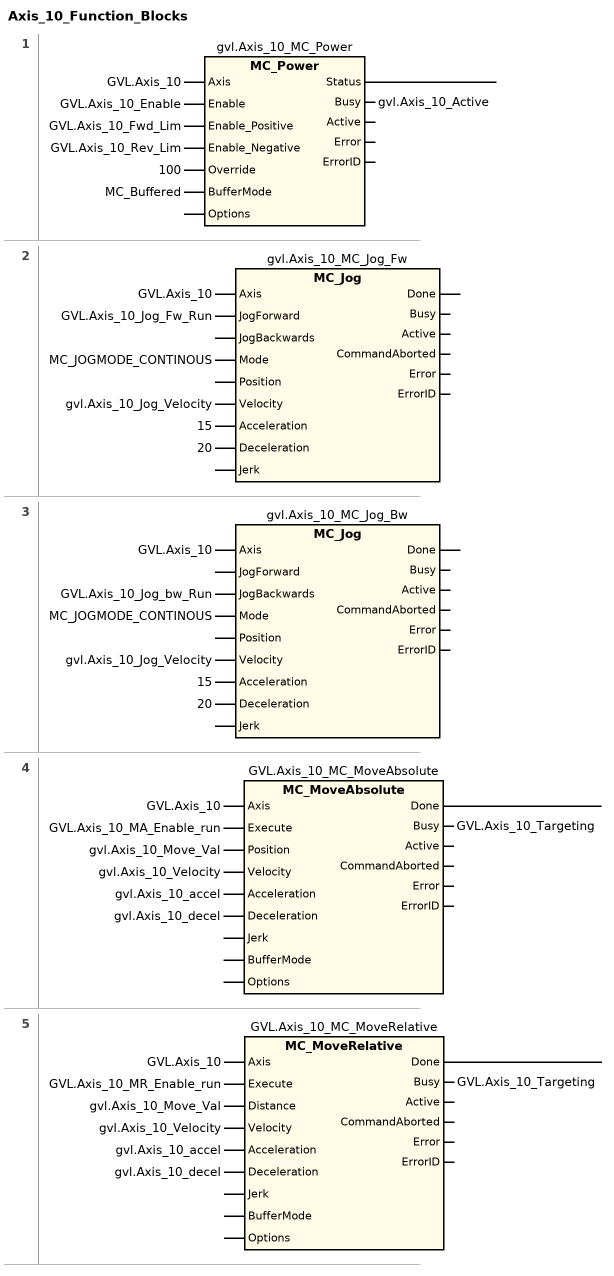
// NETWORK 1
gvl.Axis_10_MC_Power(
    Axis := GVL.Axis_10,
    Enable := GVL.Axis_10_Enable,
    Enable_Positive := GVL.Axis_10_Fwd_Lim,
    Enable_Negative := GVL.Axis_10_Rev_Lim,
    Override := 100,
    BufferMode := MC_Buffered,
    Busy => gvl.Axis_10_Active); // MC_Power

// NETWORK 2
gvl.Axis_10_MC_Jog_Fw(
    Axis := GVL.Axis_10,
    JogForward := GVL.Axis_10_Jog_Fw_Run,
    Mode := MC_JOGMODE_CONTINOUS,
    Velocity := gvl.Axis_10_Jog_Velocity,
    Acceleration := 15,
    Deceleration := 20); // MC_Jog

// NETWORK 3
gvl.Axis_10_MC_Jog_Bw(
    Axis := GVL.Axis_10,
    JogBackwards := GVL.Axis_10_Jog_bw_Run,
    Mode := MC_JOGMODE_CONTINOUS,
    Velocity := gvl.Axis_10_Jog_Velocity,
    Acceleration := 15,
    Deceleration := 20); // MC_Jog

// NETWORK 4
GVL.Axis_10_MC_MoveAbsolute(
    Axis := GVL.Axis_10,
    Execute := GVL.Axis_10_MA_Enable_run,
    Position := gvl.Axis_10_Move_Val,
    Velocity := gvl.Axis_10_Velocity,
    Acceleration := gvl.Axis_10_accel,
    Deceleration := gvl.Axis_10_decel,
    Busy => GVL.Axis_10_Targeting); // MC_MoveAbsolute

// NETWORK 5
GVL.Axis_10_MC_MoveRelative(
    Axis := GVL.Axis_10,
    Execute := GVL.Axis_10_MR_Enable_run,
    Distance := gvl.Axis_10_Move_Val,
    Velocity := gvl.Axis_10_Velocity,
    Acceleration := gvl.Axis_10_accel,
    Deceleration := gvl.Axis_10_decel,
    Busy => GVL.Axis_10_Targeting); // MC_MoveRelative

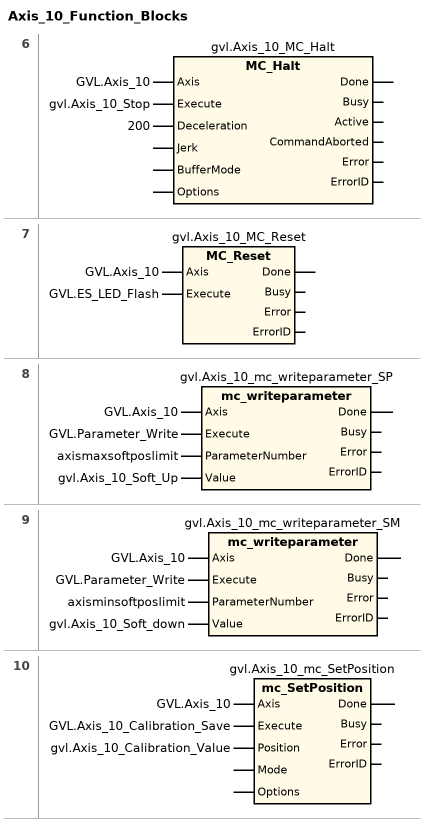
// NETWORK 6
gvl.Axis_10_MC_Halt(Axis := GVL.Axis_10, Execute := gvl.Axis_10_Stop, Deceleration := 200); // MC_Halt

// NETWORK 7
gvl.Axis_10_MC_Reset(Axis := GVL.Axis_10, Execute := GVL.ES_LED_Flash); // MC_Reset

// NETWORK 8
gvl.Axis_10_mc_writeparameter_SP(
    Axis := GVL.Axis_10,
    Execute := GVL.Parameter_Write,
    ParameterNumber := axismaxsoftposlimit,
    Value := gvl.Axis_10_Soft_Up); // mc_writeparameter

// NETWORK 9
gvl.Axis_10_mc_writeparameter_SM(
    Axis := GVL.Axis_10,
    Execute := GVL.Parameter_Write,
    ParameterNumber := axisminsoftposlimit,
    Value := gvl.Axis_10_Soft_down); // mc_writeparameter

// NETWORK 10
gvl.Axis_10_mc_SetPosition(
    Axis := GVL.Axis_10,
    Execute := GVL.Axis_10_Calibration_Save,
    Position := gvl.Axis_10_Calibration_Value); // mc_SetPosition

END_PROGRAM

// ---- POUs/Axis_10_Logic.TcPOU
PROGRAM Axis_10_Logic
VAR
	TON_0: TON;
	TON_1: TON;
	TON_2: TON;
	TON_3: TON;
	Axis_10_Velocity_Range: LREAL;
	Axis_10_Velocity_Scale: LREAL;
	Axis_10_Velocity_Raw: LREAL;
	Axis_10_Soft_Range: LREAL;
	Axis_10_Soft_Position: LREAL;
	Axis_10_Soft_Position_In_Range: LREAL;
END_VAR

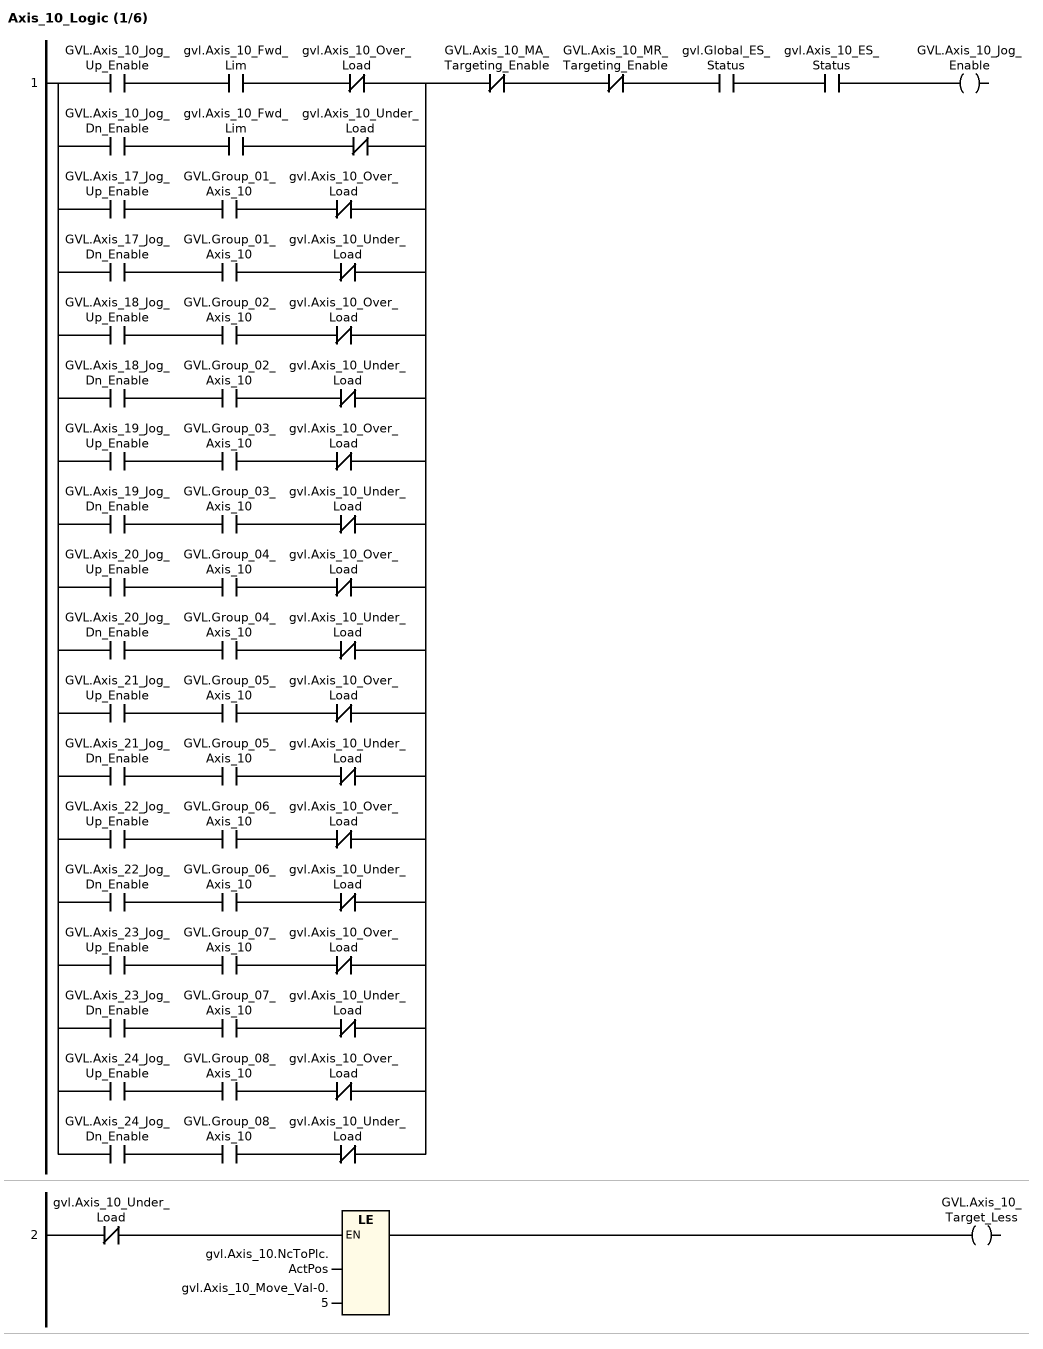
// NETWORK 1
GVL.Axis_10_Jog_Enable := (GVL.Axis_10_Jog_Up_Enable AND gvl.Axis_10_Fwd_Lim AND NOT gvl.Axis_10_Over_Load OR GVL.Axis_10_Jog_Dn_Enable AND gvl.Axis_10_Fwd_Lim AND NOT gvl.Axis_10_Under_Load OR GVL.Axis_17_Jog_Up_Enable AND GVL.Group_01_Axis_10 AND NOT gvl.Axis_10_Over_Load OR GVL.Axis_17_Jog_Dn_Enable AND GVL.Group_01_Axis_10 AND NOT gvl.Axis_10_Under_Load OR GVL.Axis_18_Jog_Up_Enable AND GVL.Group_02_Axis_10 AND NOT gvl.Axis_10_Over_Load OR GVL.Axis_18_Jog_Dn_Enable AND GVL.Group_02_Axis_10 AND NOT gvl.Axis_10_Under_Load OR GVL.Axis_19_Jog_Up_Enable AND GVL.Group_03_Axis_10 AND NOT gvl.Axis_10_Over_Load OR GVL.Axis_19_Jog_Dn_Enable AND GVL.Group_03_Axis_10 AND NOT gvl.Axis_10_Under_Load OR GVL.Axis_20_Jog_Up_Enable AND GVL.Group_04_Axis_10 AND NOT gvl.Axis_10_Over_Load OR GVL.Axis_20_Jog_Dn_Enable AND GVL.Group_04_Axis_10 AND NOT gvl.Axis_10_Under_Load OR GVL.Axis_21_Jog_Up_Enable AND GVL.Group_05_Axis_10 AND NOT gvl.Axis_10_Over_Load OR GVL.Axis_21_Jog_Dn_Enable AND GVL.Group_05_Axis_10 AND NOT gvl.Axis_10_Under_Load OR GVL.Axis_22_Jog_Up_Enable AND GVL.Group_06_Axis_10 AND NOT gvl.Axis_10_Over_Load OR GVL.Axis_22_Jog_Dn_Enable AND GVL.Group_06_Axis_10 AND NOT gvl.Axis_10_Under_Load OR GVL.Axis_23_Jog_Up_Enable AND GVL.Group_07_Axis_10 AND NOT gvl.Axis_10_Over_Load OR GVL.Axis_23_Jog_Dn_Enable AND GVL.Group_07_Axis_10 AND NOT gvl.Axis_10_Under_Load OR GVL.Axis_24_Jog_Up_Enable AND GVL.Group_08_Axis_10 AND NOT gvl.Axis_10_Over_Load OR GVL.Axis_24_Jog_Dn_Enable AND GVL.Group_08_Axis_10 AND NOT gvl.Axis_10_Under_Load) AND NOT GVL.Axis_10_MA_Targeting_Enable AND NOT GVL.Axis_10_MR_Targeting_Enable AND gvl.Global_ES_Status AND gvl.Axis_10_ES_Status;

// NETWORK 2
GVL.Axis_10_Target_Less := NOT gvl.Axis_10_Under_Load AND gvl.Axis_10.NcToPlc.ActPos <= (gvl.Axis_10_Move_Val-0.5);

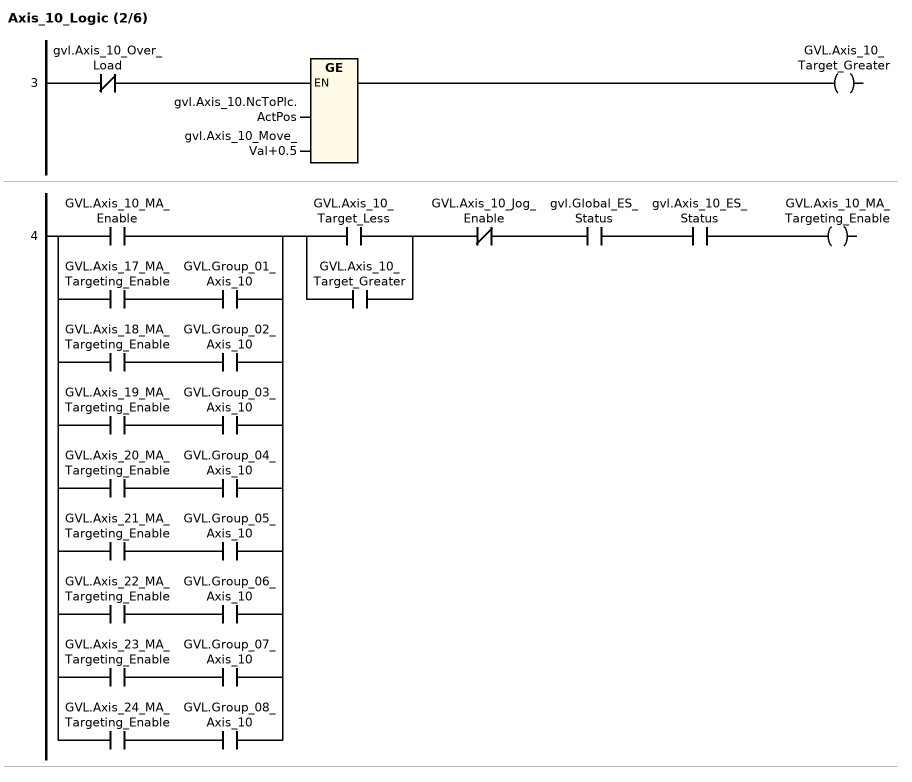
// NETWORK 3
GVL.Axis_10_Target_Greater := NOT gvl.Axis_10_Over_Load AND gvl.Axis_10.NcToPlc.ActPos >= (gvl.Axis_10_Move_Val+0.5);

// NETWORK 4
GVL.Axis_10_MA_Targeting_Enable := (GVL.Axis_10_MA_Enable OR GVL.Axis_17_MA_Targeting_Enable AND GVL.Group_01_Axis_10 OR GVL.Axis_18_MA_Targeting_Enable AND GVL.Group_02_Axis_10 OR GVL.Axis_19_MA_Targeting_Enable AND GVL.Group_03_Axis_10 OR GVL.Axis_20_MA_Targeting_Enable AND GVL.Group_04_Axis_10 OR GVL.Axis_21_MA_Targeting_Enable AND GVL.Group_05_Axis_10 OR GVL.Axis_22_MA_Targeting_Enable AND GVL.Group_06_Axis_10 OR GVL.Axis_23_MA_Targeting_Enable AND GVL.Group_07_Axis_10 OR GVL.Axis_24_MA_Targeting_Enable AND GVL.Group_08_Axis_10) AND (GVL.Axis_10_Target_Less OR GVL.Axis_10_Target_Greater) AND NOT GVL.Axis_10_Jog_Enable AND gvl.Global_ES_Status AND gvl.Axis_10_ES_Status;

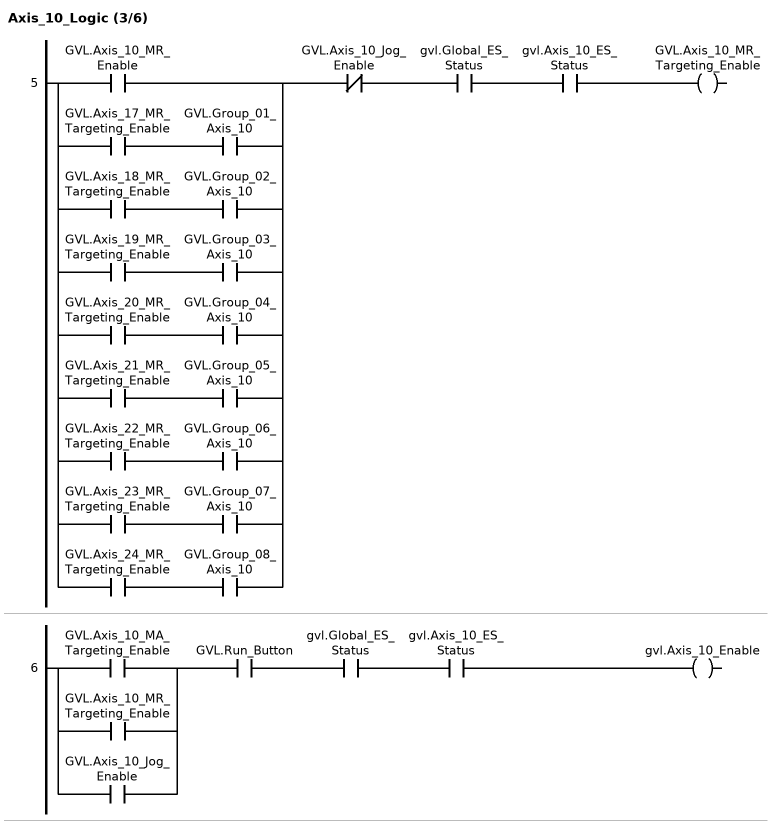
// NETWORK 5
GVL.Axis_10_MR_Targeting_Enable := (GVL.Axis_10_MR_Enable OR GVL.Axis_17_MR_Targeting_Enable AND GVL.Group_01_Axis_10 OR GVL.Axis_18_MR_Targeting_Enable AND GVL.Group_02_Axis_10 OR GVL.Axis_19_MR_Targeting_Enable AND GVL.Group_03_Axis_10 OR GVL.Axis_20_MR_Targeting_Enable AND GVL.Group_04_Axis_10 OR GVL.Axis_21_MR_Targeting_Enable AND GVL.Group_05_Axis_10 OR GVL.Axis_22_MR_Targeting_Enable AND GVL.Group_06_Axis_10 OR GVL.Axis_23_MR_Targeting_Enable AND GVL.Group_07_Axis_10 OR GVL.Axis_24_MR_Targeting_Enable AND GVL.Group_08_Axis_10) AND NOT GVL.Axis_10_Jog_Enable AND gvl.Global_ES_Status AND gvl.Axis_10_ES_Status;

// NETWORK 6
gvl.Axis_10_Enable := (GVL.Axis_10_MA_Targeting_Enable OR GVL.Axis_10_MR_Targeting_Enable OR GVL.Axis_10_Jog_Enable) AND GVL.Run_Button AND gvl.Global_ES_Status AND gvl.Axis_10_ES_Status;

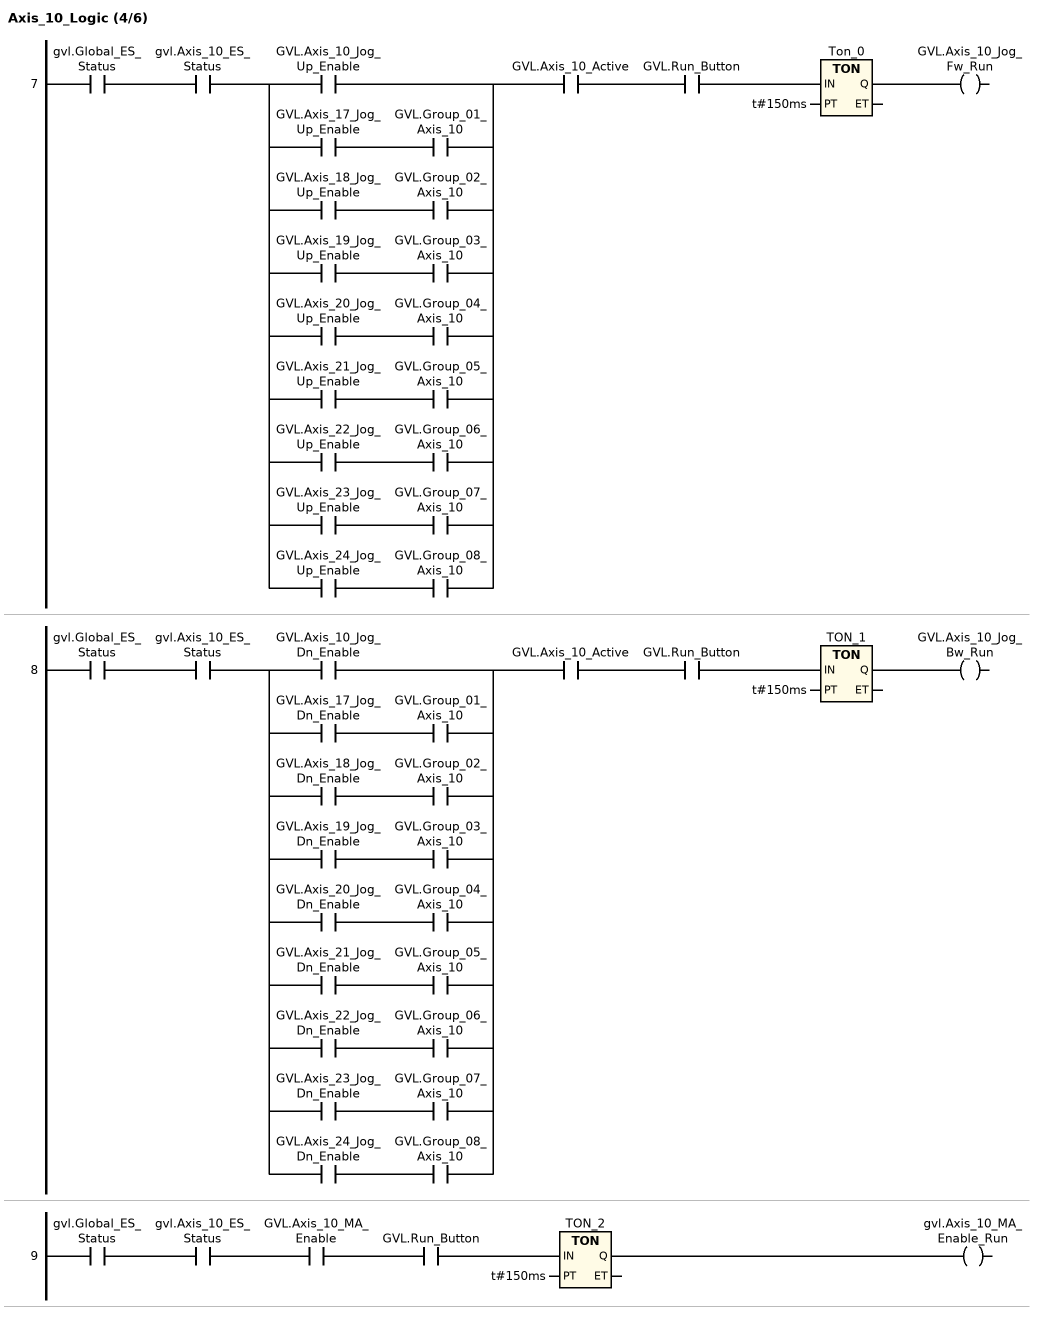
// NETWORK 7
Ton_0(IN := gvl.Global_ES_Status AND gvl.Axis_10_ES_Status AND (GVL.Axis_10_Jog_Up_Enable OR GVL.Axis_17_Jog_Up_Enable AND GVL.Group_01_Axis_10 OR GVL.Axis_18_Jog_Up_Enable AND GVL.Group_02_Axis_10 OR GVL.Axis_19_Jog_Up_Enable AND GVL.Group_03_Axis_10 OR GVL.Axis_20_Jog_Up_Enable AND GVL.Group_04_Axis_10 OR GVL.Axis_21_Jog_Up_Enable AND GVL.Group_05_Axis_10 OR GVL.Axis_22_Jog_Up_Enable AND GVL.Group_06_Axis_10 OR GVL.Axis_23_Jog_Up_Enable AND GVL.Group_07_Axis_10 OR GVL.Axis_24_Jog_Up_Enable AND GVL.Group_08_Axis_10) AND GVL.Axis_10_Active AND GVL.Run_Button, PT := t#150ms); // TON
GVL.Axis_10_Jog_Fw_Run := Ton_0.Q;

// NETWORK 8
TON_1(IN := gvl.Global_ES_Status AND gvl.Axis_10_ES_Status AND (GVL.Axis_10_Jog_Dn_Enable OR GVL.Axis_17_Jog_Dn_Enable AND GVL.Group_01_Axis_10 OR GVL.Axis_18_Jog_Dn_Enable AND GVL.Group_02_Axis_10 OR GVL.Axis_19_Jog_Dn_Enable AND GVL.Group_03_Axis_10 OR GVL.Axis_20_Jog_Dn_Enable AND GVL.Group_04_Axis_10 OR GVL.Axis_21_Jog_Dn_Enable AND GVL.Group_05_Axis_10 OR GVL.Axis_22_Jog_Dn_Enable AND GVL.Group_06_Axis_10 OR GVL.Axis_23_Jog_Dn_Enable AND GVL.Group_07_Axis_10 OR GVL.Axis_24_Jog_Dn_Enable AND GVL.Group_08_Axis_10) AND GVL.Axis_10_Active AND GVL.Run_Button, PT := t#150ms); // TON
GVL.Axis_10_Jog_Bw_Run := TON_1.Q;

// NETWORK 9
TON_2(IN := gvl.Global_ES_Status AND gvl.Axis_10_ES_Status AND GVL.Axis_10_MA_Enable AND GVL.Run_Button, PT := t#150ms); // TON
gvl.Axis_10_MA_Enable_Run := TON_2.Q;

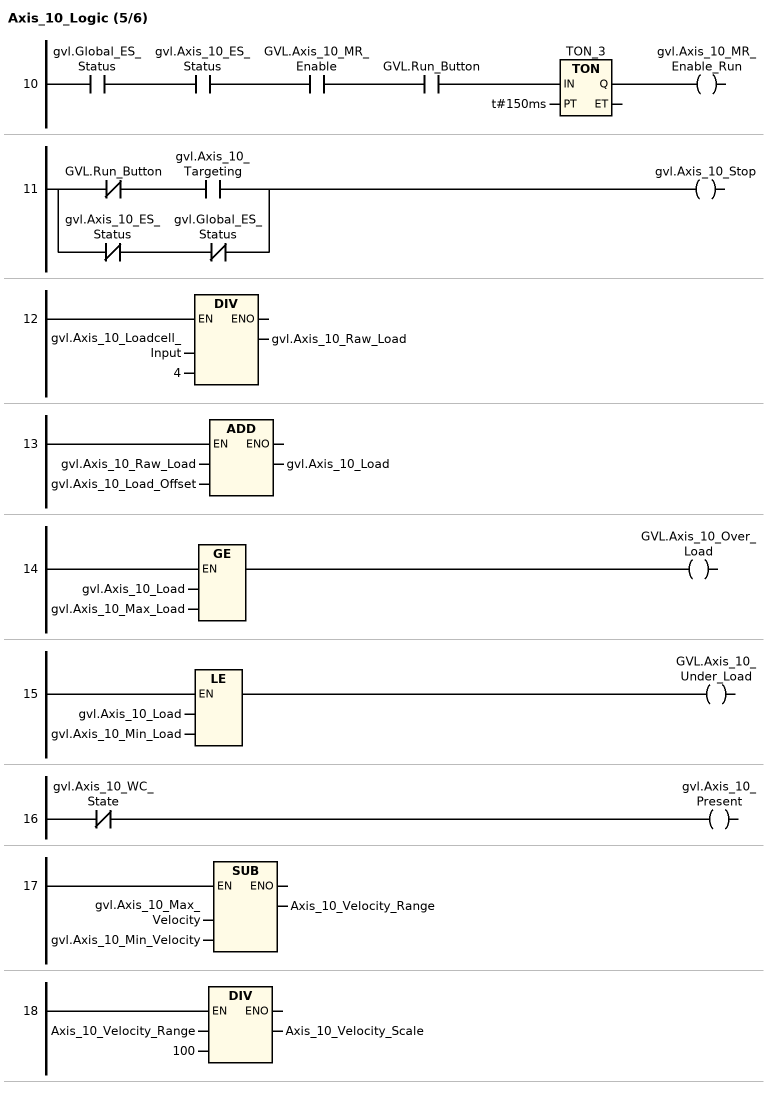
// NETWORK 10
TON_3(IN := gvl.Global_ES_Status AND gvl.Axis_10_ES_Status AND GVL.Axis_10_MR_Enable AND GVL.Run_Button, PT := t#150ms); // TON
gvl.Axis_10_MR_Enable_Run := TON_3.Q;

// NETWORK 11
gvl.Axis_10_Stop := NOT GVL.Run_Button AND gvl.Axis_10_Targeting OR NOT gvl.Axis_10_ES_Status AND NOT gvl.Global_ES_Status;

// NETWORK 12
gvl.Axis_10_Raw_Load := gvl.Axis_10_Loadcell_Input / 4;

// NETWORK 13
gvl.Axis_10_Load := gvl.Axis_10_Raw_Load + gvl.Axis_10_Load_Offset;

// NETWORK 14
GVL.Axis_10_Over_Load := gvl.Axis_10_Load >= gvl.Axis_10_Max_Load;

// NETWORK 15
GVL.Axis_10_Under_Load := gvl.Axis_10_Load <= gvl.Axis_10_Min_Load;

// NETWORK 16
gvl.Axis_10_Present := NOT gvl.Axis_10_WC_State;

// NETWORK 17
Axis_10_Velocity_Range := gvl.Axis_10_Max_Velocity - gvl.Axis_10_Min_Velocity;

// NETWORK 18
Axis_10_Velocity_Scale := Axis_10_Velocity_Range / 100;

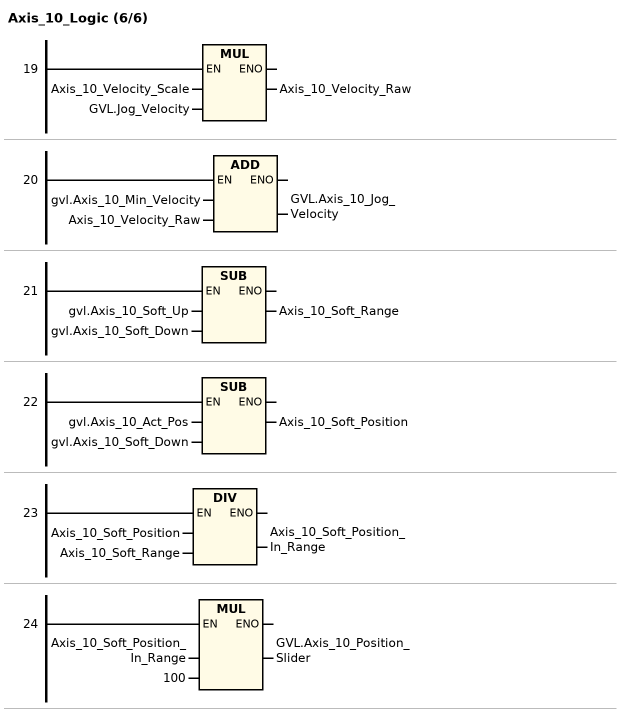
// NETWORK 19
Axis_10_Velocity_Raw := Axis_10_Velocity_Scale * GVL.Jog_Velocity;

// NETWORK 20
GVL.Axis_10_Jog_Velocity := gvl.Axis_10_Min_Velocity + Axis_10_Velocity_Raw;

// NETWORK 21
Axis_10_Soft_Range := gvl.Axis_10_Soft_Up - gvl.Axis_10_Soft_Down;

// NETWORK 22
Axis_10_Soft_Position := gvl.Axis_10_Act_Pos - gvl.Axis_10_Soft_Down;

// NETWORK 23
Axis_10_Soft_Position_In_Range := Axis_10_Soft_Position / Axis_10_Soft_Range;

// NETWORK 24
GVL.Axis_10_Position_Slider := Axis_10_Soft_Position_In_Range * 100;

END_PROGRAM

// ---- POUs/Axis_11_Function_Blocks.TcPOU
PROGRAM Axis_11_Function_Blocks
VAR
END_VAR

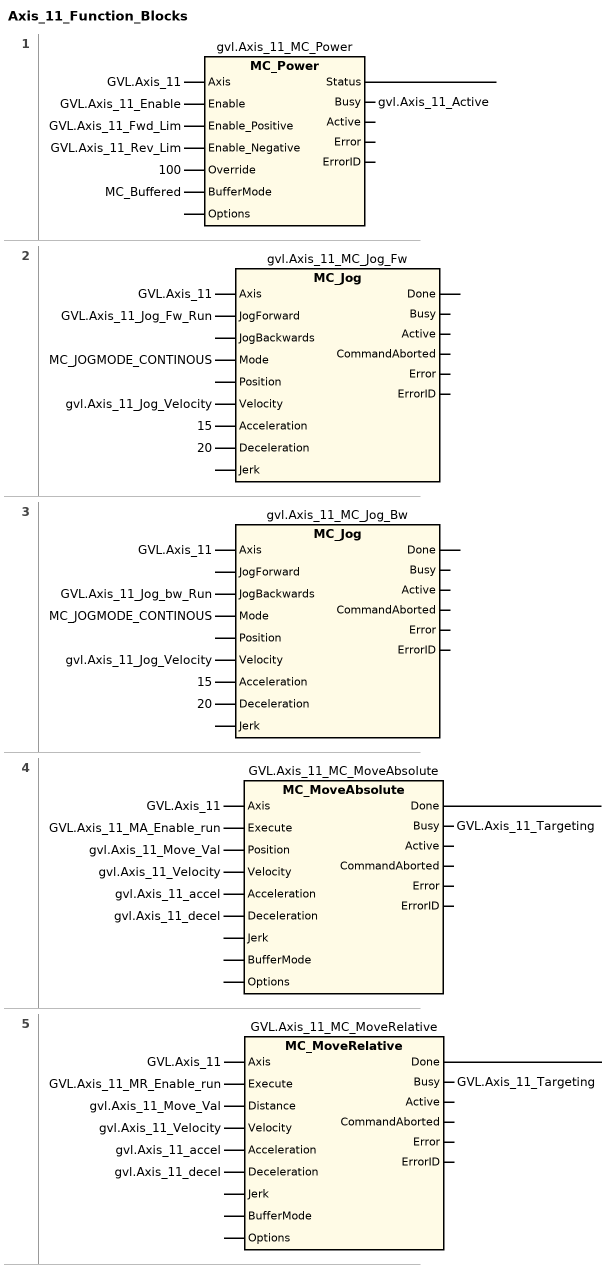
// NETWORK 1
gvl.Axis_11_MC_Power(
    Axis := GVL.Axis_11,
    Enable := GVL.Axis_11_Enable,
    Enable_Positive := GVL.Axis_11_Fwd_Lim,
    Enable_Negative := GVL.Axis_11_Rev_Lim,
    Override := 100,
    BufferMode := MC_Buffered,
    Busy => gvl.Axis_11_Active); // MC_Power

// NETWORK 2
gvl.Axis_11_MC_Jog_Fw(
    Axis := GVL.Axis_11,
    JogForward := GVL.Axis_11_Jog_Fw_Run,
    Mode := MC_JOGMODE_CONTINOUS,
    Velocity := gvl.Axis_11_Jog_Velocity,
    Acceleration := 15,
    Deceleration := 20); // MC_Jog

// NETWORK 3
gvl.Axis_11_MC_Jog_Bw(
    Axis := GVL.Axis_11,
    JogBackwards := GVL.Axis_11_Jog_bw_Run,
    Mode := MC_JOGMODE_CONTINOUS,
    Velocity := gvl.Axis_11_Jog_Velocity,
    Acceleration := 15,
    Deceleration := 20); // MC_Jog

// NETWORK 4
GVL.Axis_11_MC_MoveAbsolute(
    Axis := GVL.Axis_11,
    Execute := GVL.Axis_11_MA_Enable_run,
    Position := gvl.Axis_11_Move_Val,
    Velocity := gvl.Axis_11_Velocity,
    Acceleration := gvl.Axis_11_accel,
    Deceleration := gvl.Axis_11_decel,
    Busy => GVL.Axis_11_Targeting); // MC_MoveAbsolute

// NETWORK 5
GVL.Axis_11_MC_MoveRelative(
    Axis := GVL.Axis_11,
    Execute := GVL.Axis_11_MR_Enable_run,
    Distance := gvl.Axis_11_Move_Val,
    Velocity := gvl.Axis_11_Velocity,
    Acceleration := gvl.Axis_11_accel,
    Deceleration := gvl.Axis_11_decel,
    Busy => GVL.Axis_11_Targeting); // MC_MoveRelative

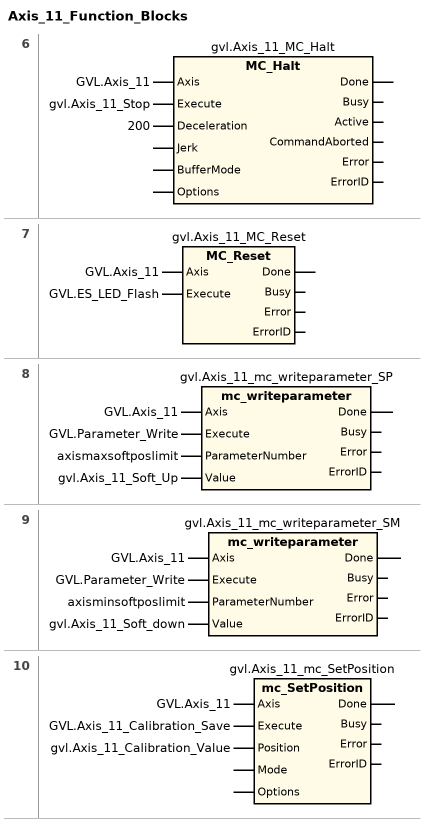
// NETWORK 6
gvl.Axis_11_MC_Halt(Axis := GVL.Axis_11, Execute := gvl.Axis_11_Stop, Deceleration := 200); // MC_Halt

// NETWORK 7
gvl.Axis_11_MC_Reset(Axis := GVL.Axis_11, Execute := GVL.ES_LED_Flash); // MC_Reset

// NETWORK 8
gvl.Axis_11_mc_writeparameter_SP(
    Axis := GVL.Axis_11,
    Execute := GVL.Parameter_Write,
    ParameterNumber := axismaxsoftposlimit,
    Value := gvl.Axis_11_Soft_Up); // mc_writeparameter

// NETWORK 9
gvl.Axis_11_mc_writeparameter_SM(
    Axis := GVL.Axis_11,
    Execute := GVL.Parameter_Write,
    ParameterNumber := axisminsoftposlimit,
    Value := gvl.Axis_11_Soft_down); // mc_writeparameter

// NETWORK 10
gvl.Axis_11_mc_SetPosition(
    Axis := GVL.Axis_11,
    Execute := GVL.Axis_11_Calibration_Save,
    Position := gvl.Axis_11_Calibration_Value); // mc_SetPosition

END_PROGRAM

// ---- POUs/Axis_11_Logic.TcPOU
PROGRAM Axis_11_Logic
VAR
	TON_0: TON;
	TON_1: TON;
	TON_2: TON;
	TON_3: TON;
	Axis_11_Velocity_Range: LREAL;
	Axis_11_Velocity_Scale: LREAL;
	Axis_11_Velocity_Raw: LREAL;
	Axis_11_Soft_Range: LREAL;
	Axis_11_Soft_Position: LREAL;
	Axis_11_Soft_Position_In_Range: LREAL;
END_VAR

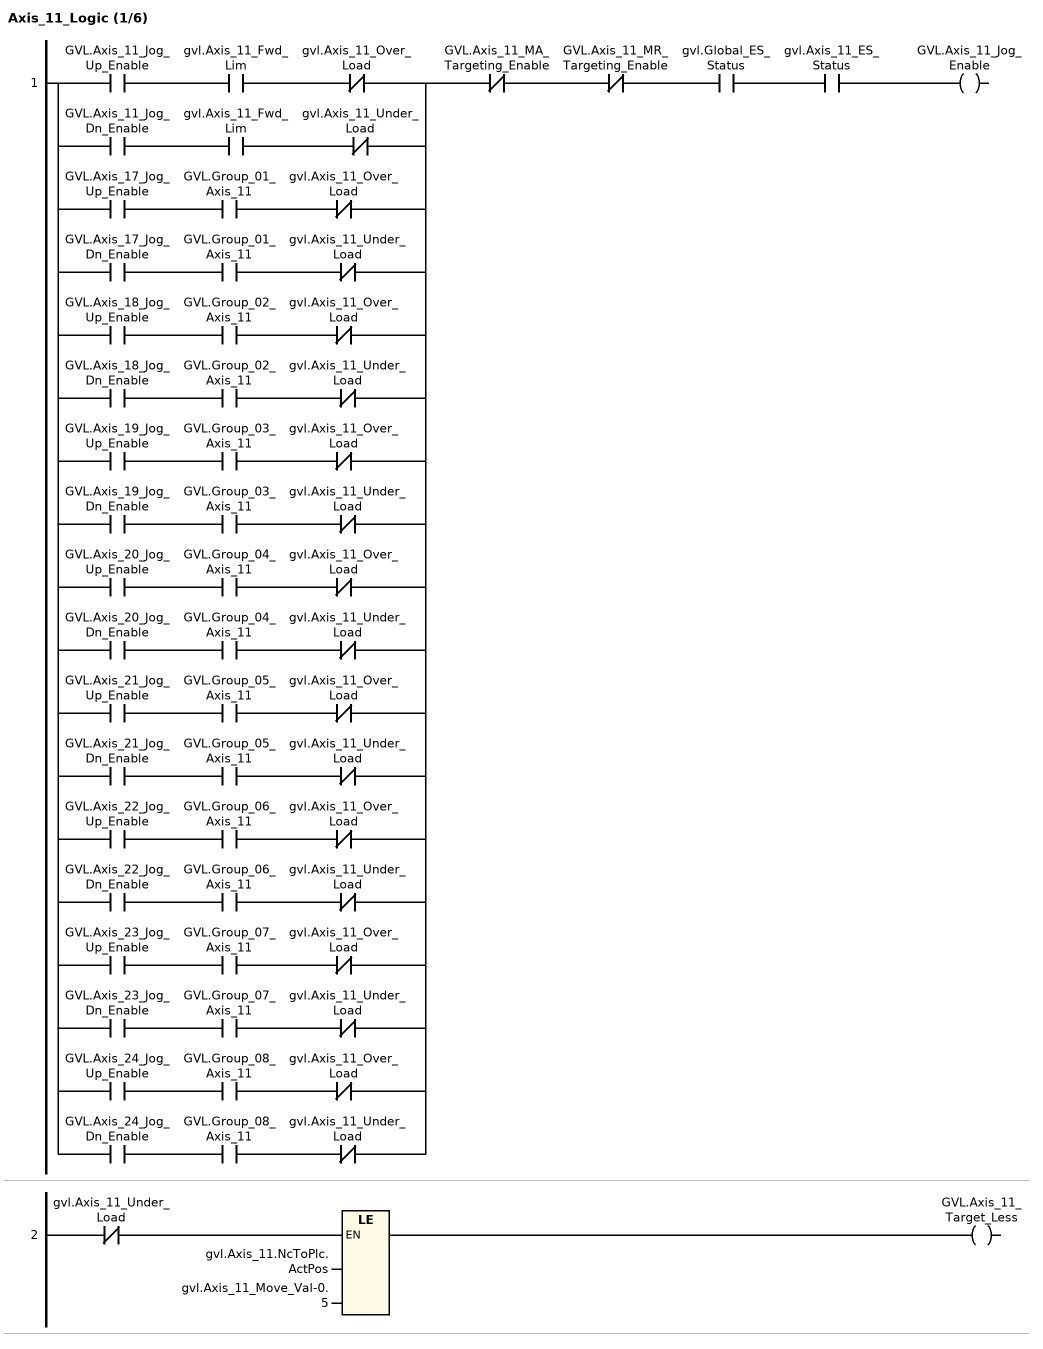
// NETWORK 1
GVL.Axis_11_Jog_Enable := (GVL.Axis_11_Jog_Up_Enable AND gvl.Axis_11_Fwd_Lim AND NOT gvl.Axis_11_Over_Load OR GVL.Axis_11_Jog_Dn_Enable AND gvl.Axis_11_Fwd_Lim AND NOT gvl.Axis_11_Under_Load OR GVL.Axis_17_Jog_Up_Enable AND GVL.Group_01_Axis_11 AND NOT gvl.Axis_11_Over_Load OR GVL.Axis_17_Jog_Dn_Enable AND GVL.Group_01_Axis_11 AND NOT gvl.Axis_11_Under_Load OR GVL.Axis_18_Jog_Up_Enable AND GVL.Group_02_Axis_11 AND NOT gvl.Axis_11_Over_Load OR GVL.Axis_18_Jog_Dn_Enable AND GVL.Group_02_Axis_11 AND NOT gvl.Axis_11_Under_Load OR GVL.Axis_19_Jog_Up_Enable AND GVL.Group_03_Axis_11 AND NOT gvl.Axis_11_Over_Load OR GVL.Axis_19_Jog_Dn_Enable AND GVL.Group_03_Axis_11 AND NOT gvl.Axis_11_Under_Load OR GVL.Axis_20_Jog_Up_Enable AND GVL.Group_04_Axis_11 AND NOT gvl.Axis_11_Over_Load OR GVL.Axis_20_Jog_Dn_Enable AND GVL.Group_04_Axis_11 AND NOT gvl.Axis_11_Under_Load OR GVL.Axis_21_Jog_Up_Enable AND GVL.Group_05_Axis_11 AND NOT gvl.Axis_11_Over_Load OR GVL.Axis_21_Jog_Dn_Enable AND GVL.Group_05_Axis_11 AND NOT gvl.Axis_11_Under_Load OR GVL.Axis_22_Jog_Up_Enable AND GVL.Group_06_Axis_11 AND NOT gvl.Axis_11_Over_Load OR GVL.Axis_22_Jog_Dn_Enable AND GVL.Group_06_Axis_11 AND NOT gvl.Axis_11_Under_Load OR GVL.Axis_23_Jog_Up_Enable AND GVL.Group_07_Axis_11 AND NOT gvl.Axis_11_Over_Load OR GVL.Axis_23_Jog_Dn_Enable AND GVL.Group_07_Axis_11 AND NOT gvl.Axis_11_Under_Load OR GVL.Axis_24_Jog_Up_Enable AND GVL.Group_08_Axis_11 AND NOT gvl.Axis_11_Over_Load OR GVL.Axis_24_Jog_Dn_Enable AND GVL.Group_08_Axis_11 AND NOT gvl.Axis_11_Under_Load) AND NOT GVL.Axis_11_MA_Targeting_Enable AND NOT GVL.Axis_11_MR_Targeting_Enable AND gvl.Global_ES_Status AND gvl.Axis_11_ES_Status;

// NETWORK 2
GVL.Axis_11_Target_Less := NOT gvl.Axis_11_Under_Load AND gvl.Axis_11.NcToPlc.ActPos <= (gvl.Axis_11_Move_Val-0.5);

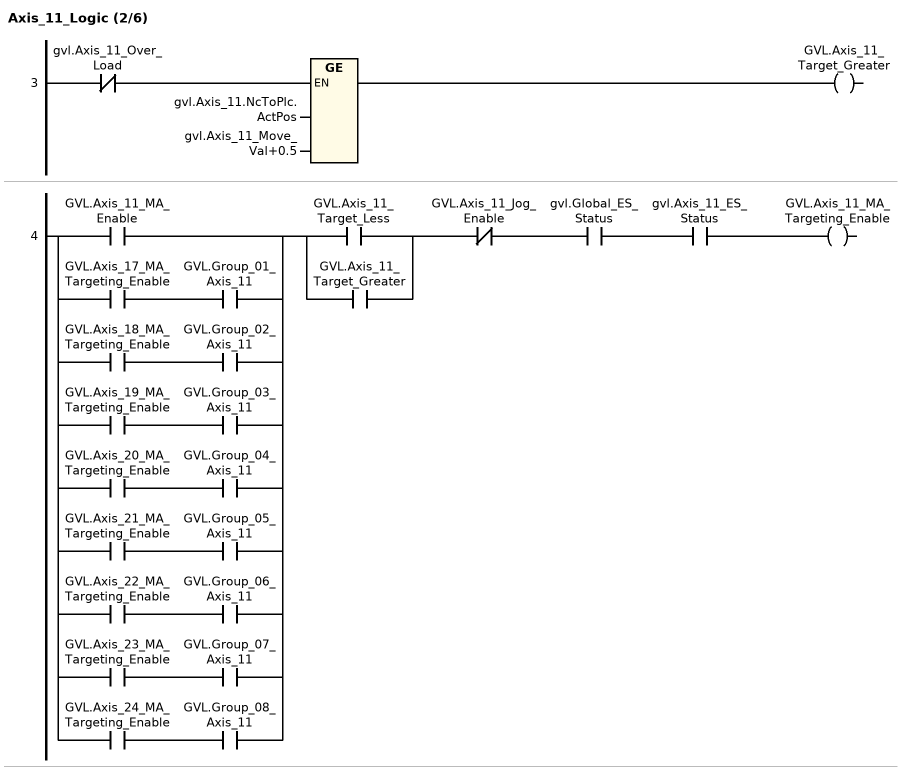
// NETWORK 3
GVL.Axis_11_Target_Greater := NOT gvl.Axis_11_Over_Load AND gvl.Axis_11.NcToPlc.ActPos >= (gvl.Axis_11_Move_Val+0.5);

// NETWORK 4
GVL.Axis_11_MA_Targeting_Enable := (GVL.Axis_11_MA_Enable OR GVL.Axis_17_MA_Targeting_Enable AND GVL.Group_01_Axis_11 OR GVL.Axis_18_MA_Targeting_Enable AND GVL.Group_02_Axis_11 OR GVL.Axis_19_MA_Targeting_Enable AND GVL.Group_03_Axis_11 OR GVL.Axis_20_MA_Targeting_Enable AND GVL.Group_04_Axis_11 OR GVL.Axis_21_MA_Targeting_Enable AND GVL.Group_05_Axis_11 OR GVL.Axis_22_MA_Targeting_Enable AND GVL.Group_06_Axis_11 OR GVL.Axis_23_MA_Targeting_Enable AND GVL.Group_07_Axis_11 OR GVL.Axis_24_MA_Targeting_Enable AND GVL.Group_08_Axis_11) AND (GVL.Axis_11_Target_Less OR GVL.Axis_11_Target_Greater) AND NOT GVL.Axis_11_Jog_Enable AND gvl.Global_ES_Status AND gvl.Axis_11_ES_Status;

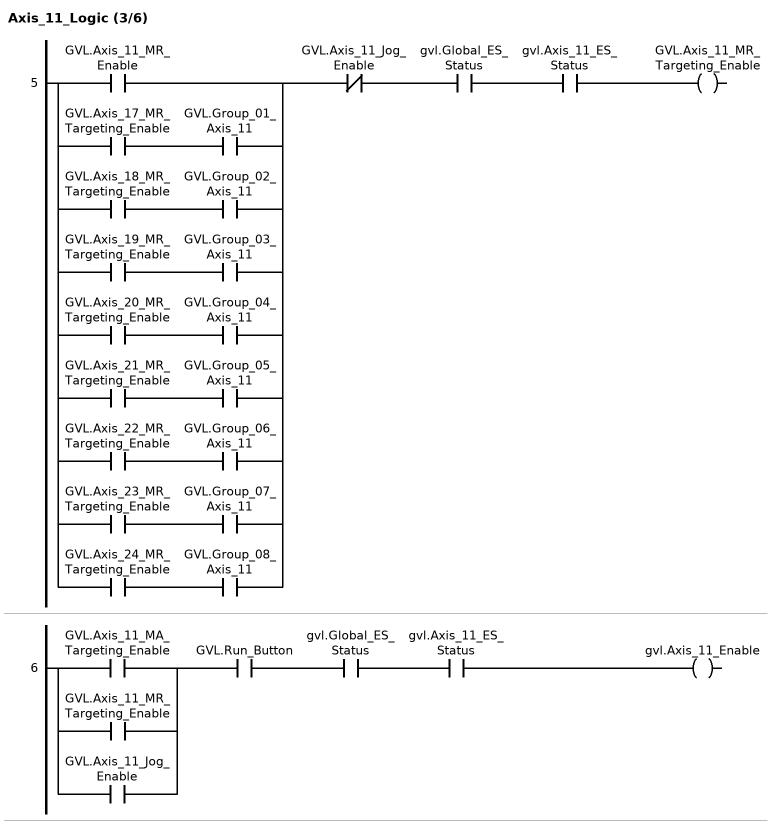
// NETWORK 5
GVL.Axis_11_MR_Targeting_Enable := (GVL.Axis_11_MR_Enable OR GVL.Axis_17_MR_Targeting_Enable AND GVL.Group_01_Axis_11 OR GVL.Axis_18_MR_Targeting_Enable AND GVL.Group_02_Axis_11 OR GVL.Axis_19_MR_Targeting_Enable AND GVL.Group_03_Axis_11 OR GVL.Axis_20_MR_Targeting_Enable AND GVL.Group_04_Axis_11 OR GVL.Axis_21_MR_Targeting_Enable AND GVL.Group_05_Axis_11 OR GVL.Axis_22_MR_Targeting_Enable AND GVL.Group_06_Axis_11 OR GVL.Axis_23_MR_Targeting_Enable AND GVL.Group_07_Axis_11 OR GVL.Axis_24_MR_Targeting_Enable AND GVL.Group_08_Axis_11) AND NOT GVL.Axis_11_Jog_Enable AND gvl.Global_ES_Status AND gvl.Axis_11_ES_Status;

// NETWORK 6
gvl.Axis_11_Enable := (GVL.Axis_11_MA_Targeting_Enable OR GVL.Axis_11_MR_Targeting_Enable OR GVL.Axis_11_Jog_Enable) AND GVL.Run_Button AND gvl.Global_ES_Status AND gvl.Axis_11_ES_Status;

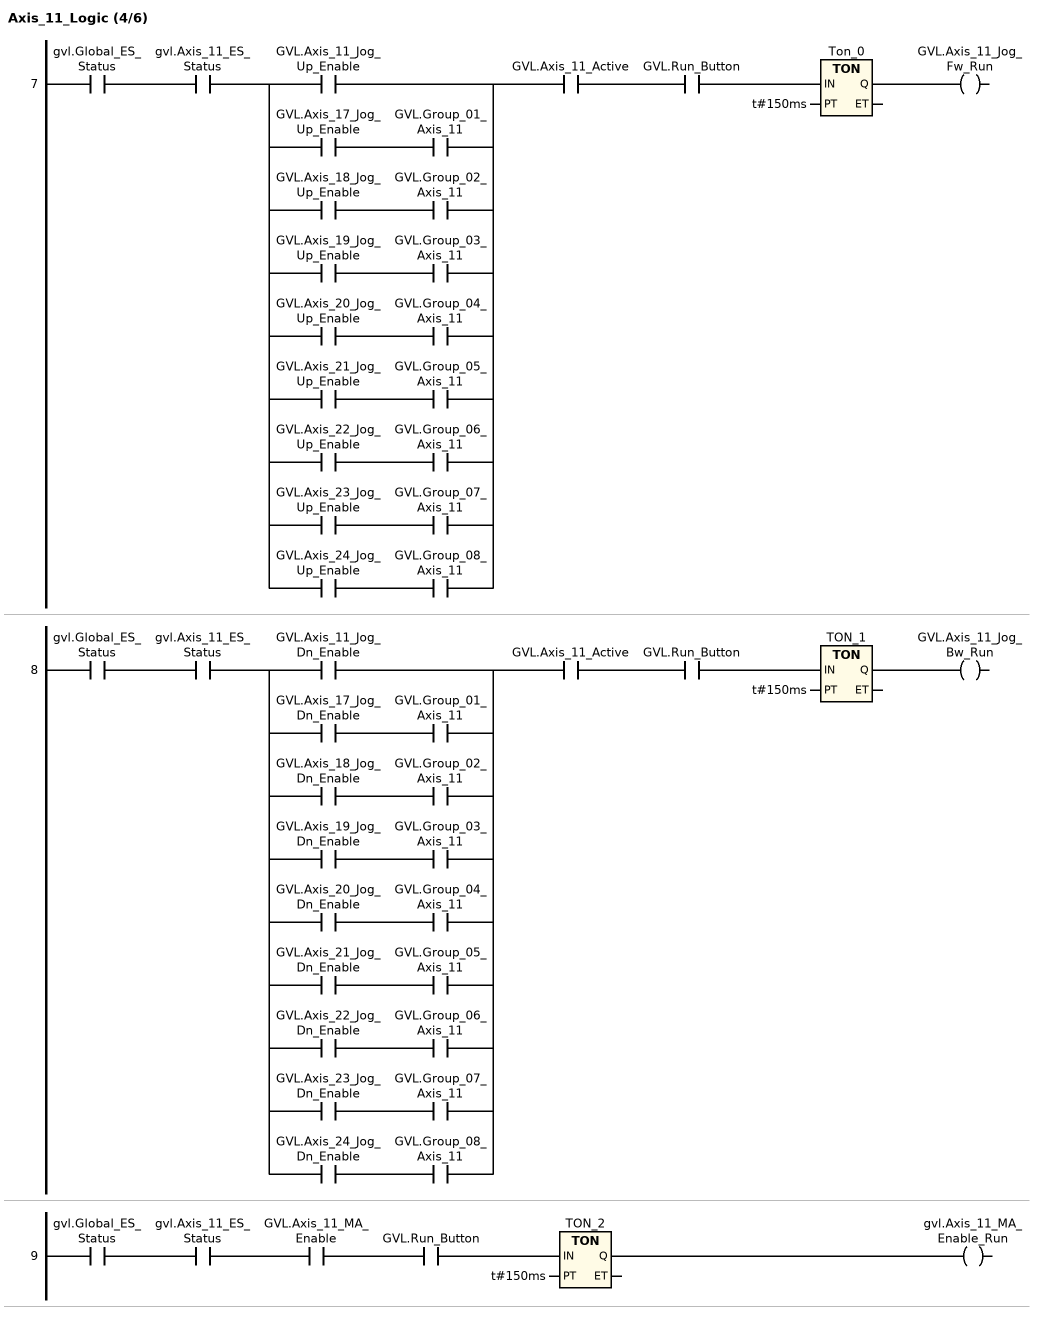
// NETWORK 7
Ton_0(IN := gvl.Global_ES_Status AND gvl.Axis_11_ES_Status AND (GVL.Axis_11_Jog_Up_Enable OR GVL.Axis_17_Jog_Up_Enable AND GVL.Group_01_Axis_11 OR GVL.Axis_18_Jog_Up_Enable AND GVL.Group_02_Axis_11 OR GVL.Axis_19_Jog_Up_Enable AND GVL.Group_03_Axis_11 OR GVL.Axis_20_Jog_Up_Enable AND GVL.Group_04_Axis_11 OR GVL.Axis_21_Jog_Up_Enable AND GVL.Group_05_Axis_11 OR GVL.Axis_22_Jog_Up_Enable AND GVL.Group_06_Axis_11 OR GVL.Axis_23_Jog_Up_Enable AND GVL.Group_07_Axis_11 OR GVL.Axis_24_Jog_Up_Enable AND GVL.Group_08_Axis_11) AND GVL.Axis_11_Active AND GVL.Run_Button, PT := t#150ms); // TON
GVL.Axis_11_Jog_Fw_Run := Ton_0.Q;

// NETWORK 8
TON_1(IN := gvl.Global_ES_Status AND gvl.Axis_11_ES_Status AND (GVL.Axis_11_Jog_Dn_Enable OR GVL.Axis_17_Jog_Dn_Enable AND GVL.Group_01_Axis_11 OR GVL.Axis_18_Jog_Dn_Enable AND GVL.Group_02_Axis_11 OR GVL.Axis_19_Jog_Dn_Enable AND GVL.Group_03_Axis_11 OR GVL.Axis_20_Jog_Dn_Enable AND GVL.Group_04_Axis_11 OR GVL.Axis_21_Jog_Dn_Enable AND GVL.Group_05_Axis_11 OR GVL.Axis_22_Jog_Dn_Enable AND GVL.Group_06_Axis_11 OR GVL.Axis_23_Jog_Dn_Enable AND GVL.Group_07_Axis_11 OR GVL.Axis_24_Jog_Dn_Enable AND GVL.Group_08_Axis_11) AND GVL.Axis_11_Active AND GVL.Run_Button, PT := t#150ms); // TON
GVL.Axis_11_Jog_Bw_Run := TON_1.Q;

// NETWORK 9
TON_2(IN := gvl.Global_ES_Status AND gvl.Axis_11_ES_Status AND GVL.Axis_11_MA_Enable AND GVL.Run_Button, PT := t#150ms); // TON
gvl.Axis_11_MA_Enable_Run := TON_2.Q;

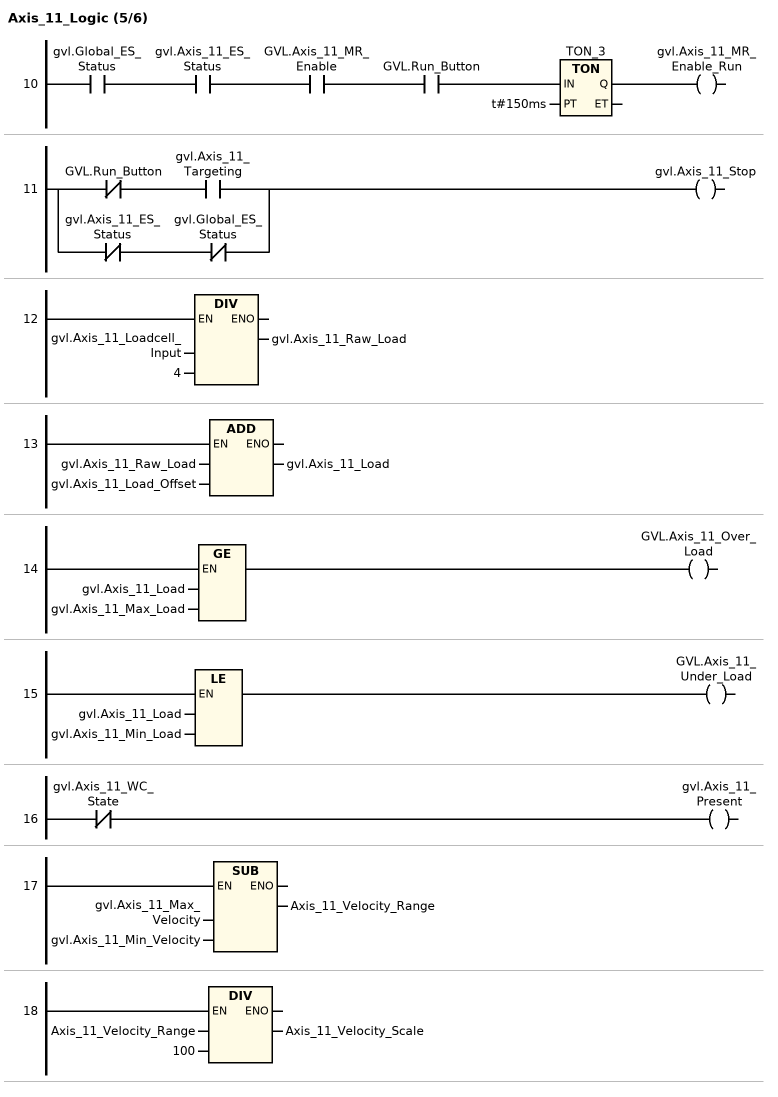
// NETWORK 10
TON_3(IN := gvl.Global_ES_Status AND gvl.Axis_11_ES_Status AND GVL.Axis_11_MR_Enable AND GVL.Run_Button, PT := t#150ms); // TON
gvl.Axis_11_MR_Enable_Run := TON_3.Q;

// NETWORK 11
gvl.Axis_11_Stop := NOT GVL.Run_Button AND gvl.Axis_11_Targeting OR NOT gvl.Axis_11_ES_Status AND NOT gvl.Global_ES_Status;

// NETWORK 12
gvl.Axis_11_Raw_Load := gvl.Axis_11_Loadcell_Input / 4;

// NETWORK 13
gvl.Axis_11_Load := gvl.Axis_11_Raw_Load + gvl.Axis_11_Load_Offset;

// NETWORK 14
GVL.Axis_11_Over_Load := gvl.Axis_11_Load >= gvl.Axis_11_Max_Load;

// NETWORK 15
GVL.Axis_11_Under_Load := gvl.Axis_11_Load <= gvl.Axis_11_Min_Load;

// NETWORK 16
gvl.Axis_11_Present := NOT gvl.Axis_11_WC_State;

// NETWORK 17
Axis_11_Velocity_Range := gvl.Axis_11_Max_Velocity - gvl.Axis_11_Min_Velocity;

// NETWORK 18
Axis_11_Velocity_Scale := Axis_11_Velocity_Range / 100;

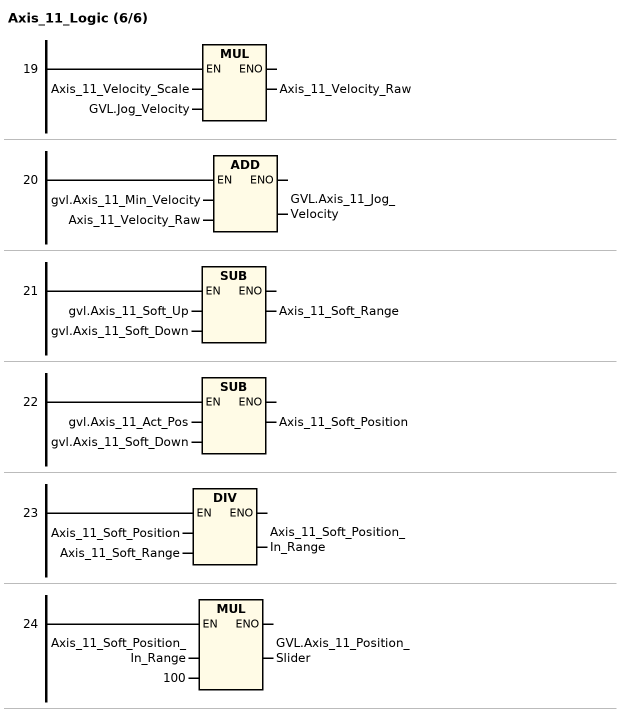
// NETWORK 19
Axis_11_Velocity_Raw := Axis_11_Velocity_Scale * GVL.Jog_Velocity;

// NETWORK 20
GVL.Axis_11_Jog_Velocity := gvl.Axis_11_Min_Velocity + Axis_11_Velocity_Raw;

// NETWORK 21
Axis_11_Soft_Range := gvl.Axis_11_Soft_Up - gvl.Axis_11_Soft_Down;

// NETWORK 22
Axis_11_Soft_Position := gvl.Axis_11_Act_Pos - gvl.Axis_11_Soft_Down;

// NETWORK 23
Axis_11_Soft_Position_In_Range := Axis_11_Soft_Position / Axis_11_Soft_Range;

// NETWORK 24
GVL.Axis_11_Position_Slider := Axis_11_Soft_Position_In_Range * 100;

END_PROGRAM

// ---- POUs/Axis_12_Function_Blocks.TcPOU
PROGRAM Axis_12_Function_Blocks
VAR
END_VAR

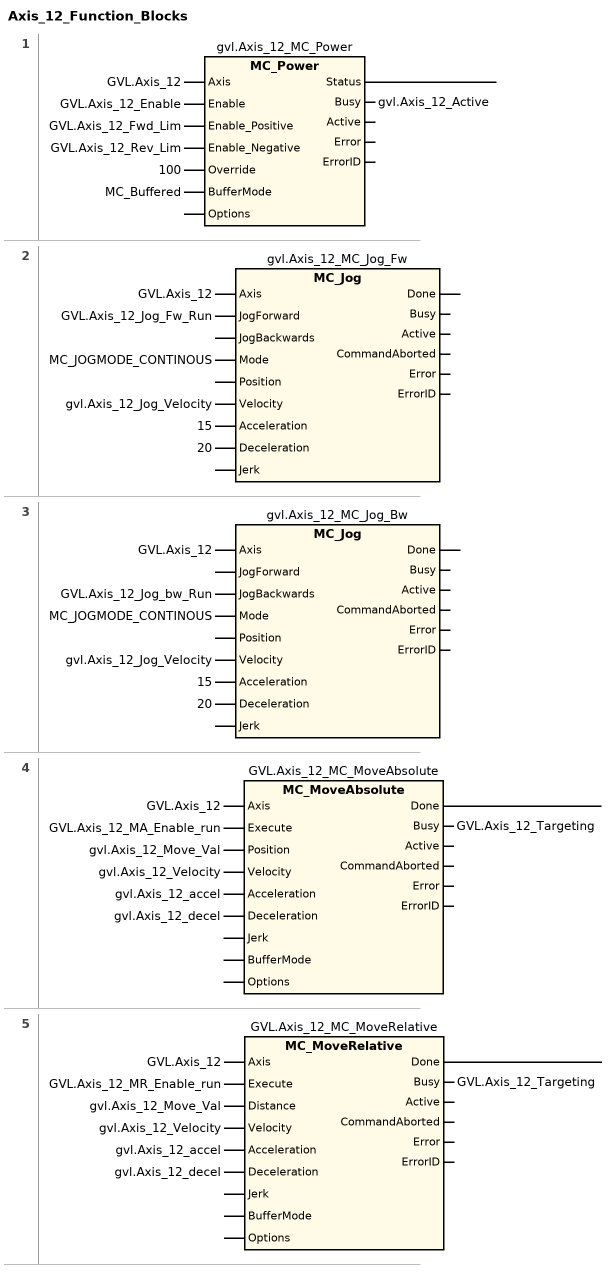
// NETWORK 1
gvl.Axis_12_MC_Power(
    Axis := GVL.Axis_12,
    Enable := GVL.Axis_12_Enable,
    Enable_Positive := GVL.Axis_12_Fwd_Lim,
    Enable_Negative := GVL.Axis_12_Rev_Lim,
    Override := 100,
    BufferMode := MC_Buffered,
    Busy => gvl.Axis_12_Active); // MC_Power

// NETWORK 2
gvl.Axis_12_MC_Jog_Fw(
    Axis := GVL.Axis_12,
    JogForward := GVL.Axis_12_Jog_Fw_Run,
    Mode := MC_JOGMODE_CONTINOUS,
    Velocity := gvl.Axis_12_Jog_Velocity,
    Acceleration := 15,
    Deceleration := 20); // MC_Jog

// NETWORK 3
gvl.Axis_12_MC_Jog_Bw(
    Axis := GVL.Axis_12,
    JogBackwards := GVL.Axis_12_Jog_bw_Run,
    Mode := MC_JOGMODE_CONTINOUS,
    Velocity := gvl.Axis_12_Jog_Velocity,
    Acceleration := 15,
    Deceleration := 20); // MC_Jog

// NETWORK 4
GVL.Axis_12_MC_MoveAbsolute(
    Axis := GVL.Axis_12,
    Execute := GVL.Axis_12_MA_Enable_run,
    Position := gvl.Axis_12_Move_Val,
    Velocity := gvl.Axis_12_Velocity,
    Acceleration := gvl.Axis_12_accel,
    Deceleration := gvl.Axis_12_decel,
    Busy => GVL.Axis_12_Targeting); // MC_MoveAbsolute

// NETWORK 5
GVL.Axis_12_MC_MoveRelative(
    Axis := GVL.Axis_12,
    Execute := GVL.Axis_12_MR_Enable_run,
    Distance := gvl.Axis_12_Move_Val,
    Velocity := gvl.Axis_12_Velocity,
    Acceleration := gvl.Axis_12_accel,
    Deceleration := gvl.Axis_12_decel,
    Busy => GVL.Axis_12_Targeting); // MC_MoveRelative

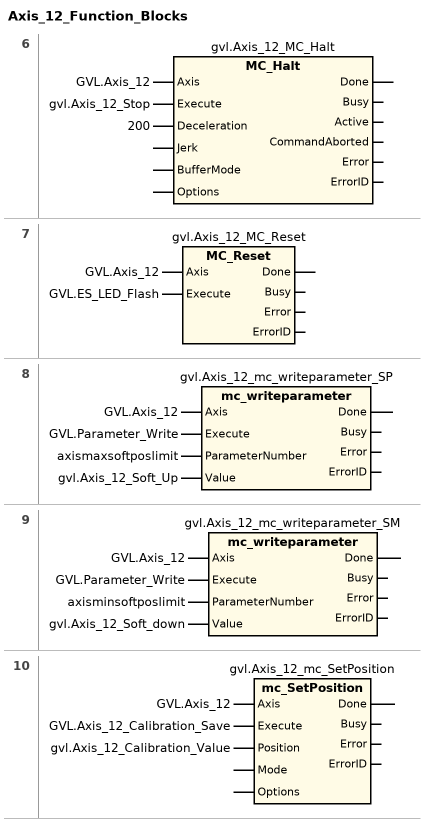
// NETWORK 6
gvl.Axis_12_MC_Halt(Axis := GVL.Axis_12, Execute := gvl.Axis_12_Stop, Deceleration := 200); // MC_Halt

// NETWORK 7
gvl.Axis_12_MC_Reset(Axis := GVL.Axis_12, Execute := GVL.ES_LED_Flash); // MC_Reset

// NETWORK 8
gvl.Axis_12_mc_writeparameter_SP(
    Axis := GVL.Axis_12,
    Execute := GVL.Parameter_Write,
    ParameterNumber := axismaxsoftposlimit,
    Value := gvl.Axis_12_Soft_Up); // mc_writeparameter

// NETWORK 9
gvl.Axis_12_mc_writeparameter_SM(
    Axis := GVL.Axis_12,
    Execute := GVL.Parameter_Write,
    ParameterNumber := axisminsoftposlimit,
    Value := gvl.Axis_12_Soft_down); // mc_writeparameter

// NETWORK 10
gvl.Axis_12_mc_SetPosition(
    Axis := GVL.Axis_12,
    Execute := GVL.Axis_12_Calibration_Save,
    Position := gvl.Axis_12_Calibration_Value); // mc_SetPosition

END_PROGRAM

// ---- POUs/Axis_12_Logic.TcPOU
PROGRAM Axis_12_Logic
VAR
	TON_0: TON;
	TON_1: TON;
	TON_2: TON;
	TON_3: TON;
	Axis_12_Velocity_Range: LREAL;
	Axis_12_Velocity_Scale: LREAL;
	Axis_12_Velocity_Raw: LREAL;
	Axis_12_Soft_Range: LREAL;
	Axis_12_Soft_Position: LREAL;
	Axis_12_Soft_Position_In_Range: LREAL;
END_VAR

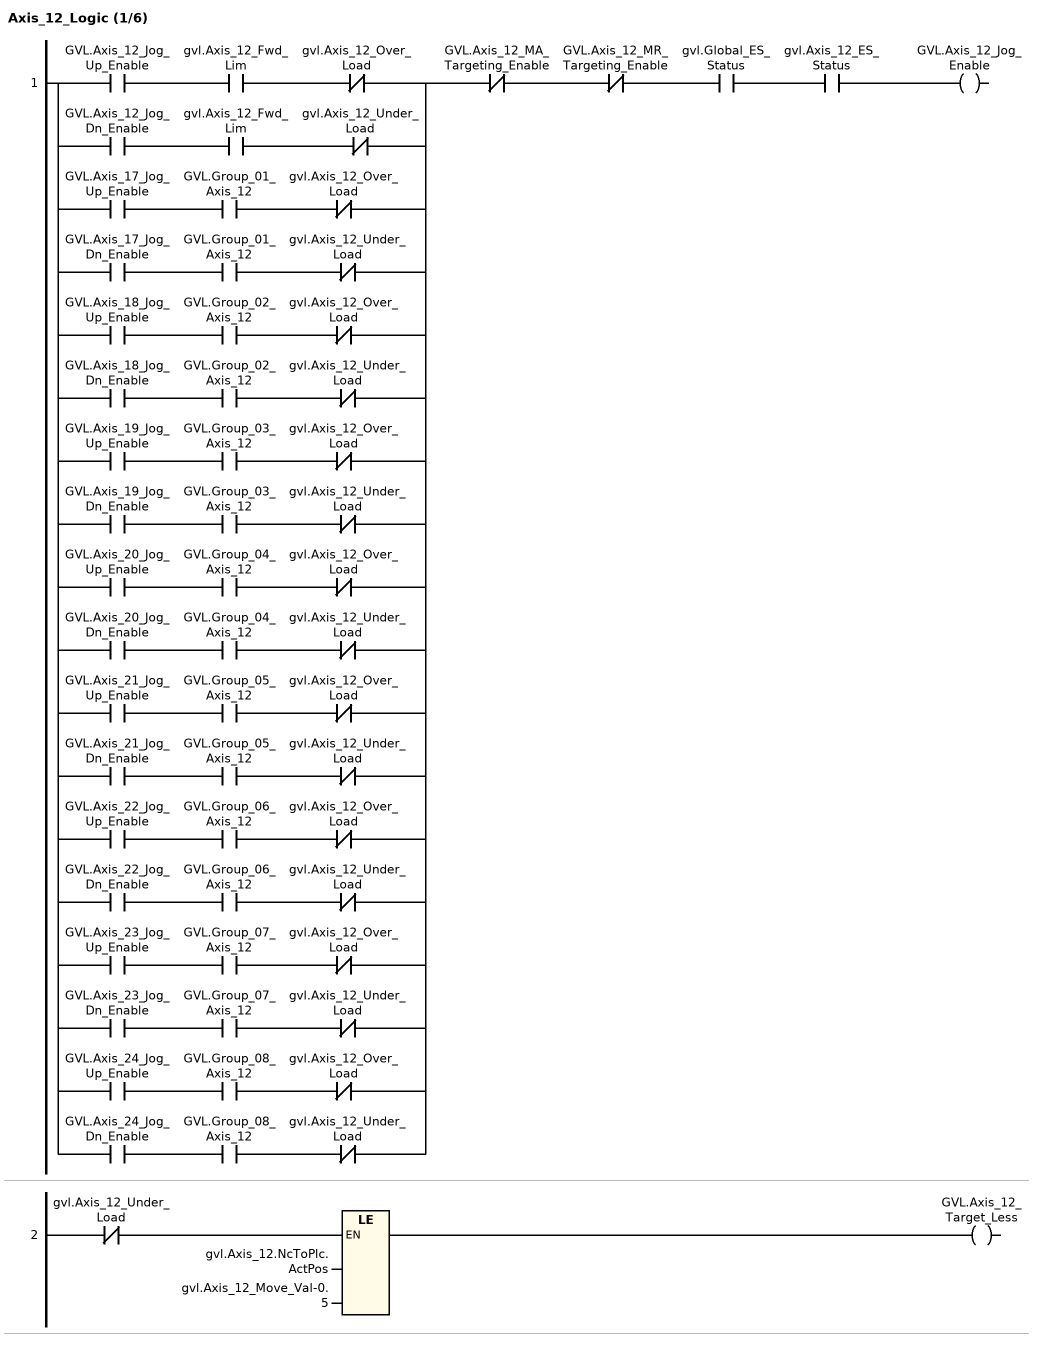
// NETWORK 1
GVL.Axis_12_Jog_Enable := (GVL.Axis_12_Jog_Up_Enable AND gvl.Axis_12_Fwd_Lim AND NOT gvl.Axis_12_Over_Load OR GVL.Axis_12_Jog_Dn_Enable AND gvl.Axis_12_Fwd_Lim AND NOT gvl.Axis_12_Under_Load OR GVL.Axis_17_Jog_Up_Enable AND GVL.Group_01_Axis_12 AND NOT gvl.Axis_12_Over_Load OR GVL.Axis_17_Jog_Dn_Enable AND GVL.Group_01_Axis_12 AND NOT gvl.Axis_12_Under_Load OR GVL.Axis_18_Jog_Up_Enable AND GVL.Group_02_Axis_12 AND NOT gvl.Axis_12_Over_Load OR GVL.Axis_18_Jog_Dn_Enable AND GVL.Group_02_Axis_12 AND NOT gvl.Axis_12_Under_Load OR GVL.Axis_19_Jog_Up_Enable AND GVL.Group_03_Axis_12 AND NOT gvl.Axis_12_Over_Load OR GVL.Axis_19_Jog_Dn_Enable AND GVL.Group_03_Axis_12 AND NOT gvl.Axis_12_Under_Load OR GVL.Axis_20_Jog_Up_Enable AND GVL.Group_04_Axis_12 AND NOT gvl.Axis_12_Over_Load OR GVL.Axis_20_Jog_Dn_Enable AND GVL.Group_04_Axis_12 AND NOT gvl.Axis_12_Under_Load OR GVL.Axis_21_Jog_Up_Enable AND GVL.Group_05_Axis_12 AND NOT gvl.Axis_12_Over_Load OR GVL.Axis_21_Jog_Dn_Enable AND GVL.Group_05_Axis_12 AND NOT gvl.Axis_12_Under_Load OR GVL.Axis_22_Jog_Up_Enable AND GVL.Group_06_Axis_12 AND NOT gvl.Axis_12_Over_Load OR GVL.Axis_22_Jog_Dn_Enable AND GVL.Group_06_Axis_12 AND NOT gvl.Axis_12_Under_Load OR GVL.Axis_23_Jog_Up_Enable AND GVL.Group_07_Axis_12 AND NOT gvl.Axis_12_Over_Load OR GVL.Axis_23_Jog_Dn_Enable AND GVL.Group_07_Axis_12 AND NOT gvl.Axis_12_Under_Load OR GVL.Axis_24_Jog_Up_Enable AND GVL.Group_08_Axis_12 AND NOT gvl.Axis_12_Over_Load OR GVL.Axis_24_Jog_Dn_Enable AND GVL.Group_08_Axis_12 AND NOT gvl.Axis_12_Under_Load) AND NOT GVL.Axis_12_MA_Targeting_Enable AND NOT GVL.Axis_12_MR_Targeting_Enable AND gvl.Global_ES_Status AND gvl.Axis_12_ES_Status;

// NETWORK 2
GVL.Axis_12_Target_Less := NOT gvl.Axis_12_Under_Load AND gvl.Axis_12.NcToPlc.ActPos <= (gvl.Axis_12_Move_Val-0.5);

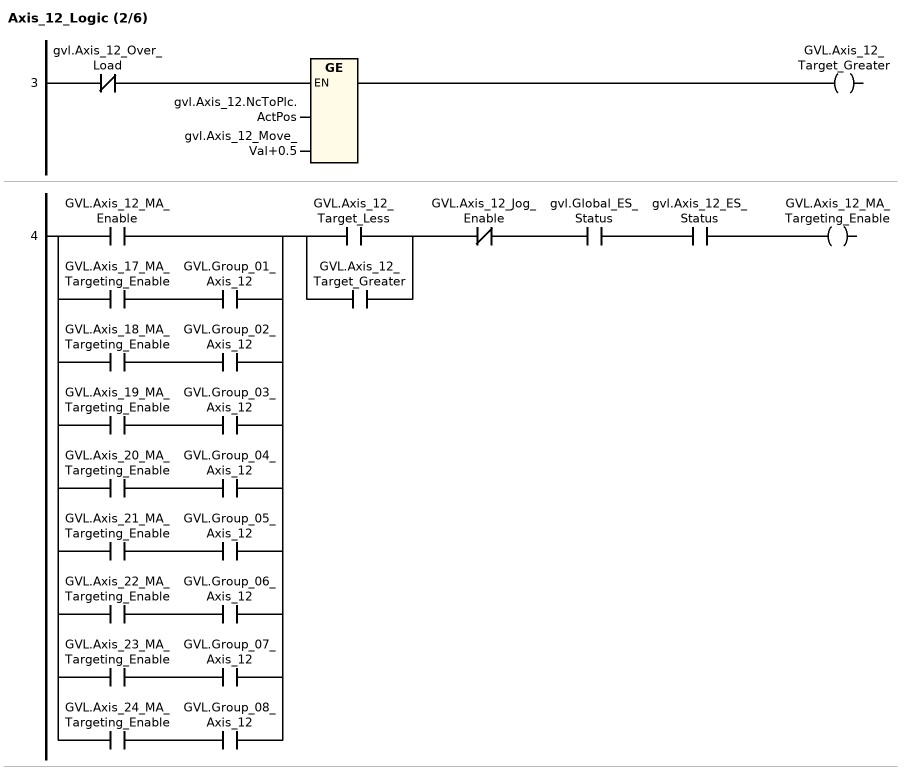
// NETWORK 3
GVL.Axis_12_Target_Greater := NOT gvl.Axis_12_Over_Load AND gvl.Axis_12.NcToPlc.ActPos >= (gvl.Axis_12_Move_Val+0.5);

// NETWORK 4
GVL.Axis_12_MA_Targeting_Enable := (GVL.Axis_12_MA_Enable OR GVL.Axis_17_MA_Targeting_Enable AND GVL.Group_01_Axis_12 OR GVL.Axis_18_MA_Targeting_Enable AND GVL.Group_02_Axis_12 OR GVL.Axis_19_MA_Targeting_Enable AND GVL.Group_03_Axis_12 OR GVL.Axis_20_MA_Targeting_Enable AND GVL.Group_04_Axis_12 OR GVL.Axis_21_MA_Targeting_Enable AND GVL.Group_05_Axis_12 OR GVL.Axis_22_MA_Targeting_Enable AND GVL.Group_06_Axis_12 OR GVL.Axis_23_MA_Targeting_Enable AND GVL.Group_07_Axis_12 OR GVL.Axis_24_MA_Targeting_Enable AND GVL.Group_08_Axis_12) AND (GVL.Axis_12_Target_Less OR GVL.Axis_12_Target_Greater) AND NOT GVL.Axis_12_Jog_Enable AND gvl.Global_ES_Status AND gvl.Axis_12_ES_Status;

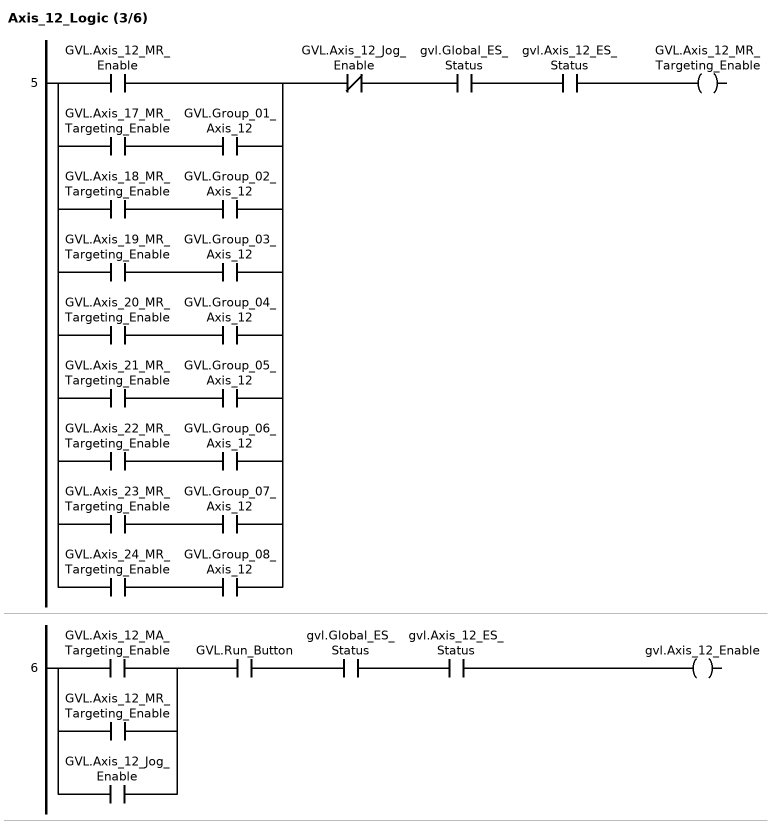
// NETWORK 5
GVL.Axis_12_MR_Targeting_Enable := (GVL.Axis_12_MR_Enable OR GVL.Axis_17_MR_Targeting_Enable AND GVL.Group_01_Axis_12 OR GVL.Axis_18_MR_Targeting_Enable AND GVL.Group_02_Axis_12 OR GVL.Axis_19_MR_Targeting_Enable AND GVL.Group_03_Axis_12 OR GVL.Axis_20_MR_Targeting_Enable AND GVL.Group_04_Axis_12 OR GVL.Axis_21_MR_Targeting_Enable AND GVL.Group_05_Axis_12 OR GVL.Axis_22_MR_Targeting_Enable AND GVL.Group_06_Axis_12 OR GVL.Axis_23_MR_Targeting_Enable AND GVL.Group_07_Axis_12 OR GVL.Axis_24_MR_Targeting_Enable AND GVL.Group_08_Axis_12) AND NOT GVL.Axis_12_Jog_Enable AND gvl.Global_ES_Status AND gvl.Axis_12_ES_Status;

// NETWORK 6
gvl.Axis_12_Enable := (GVL.Axis_12_MA_Targeting_Enable OR GVL.Axis_12_MR_Targeting_Enable OR GVL.Axis_12_Jog_Enable) AND GVL.Run_Button AND gvl.Global_ES_Status AND gvl.Axis_12_ES_Status;

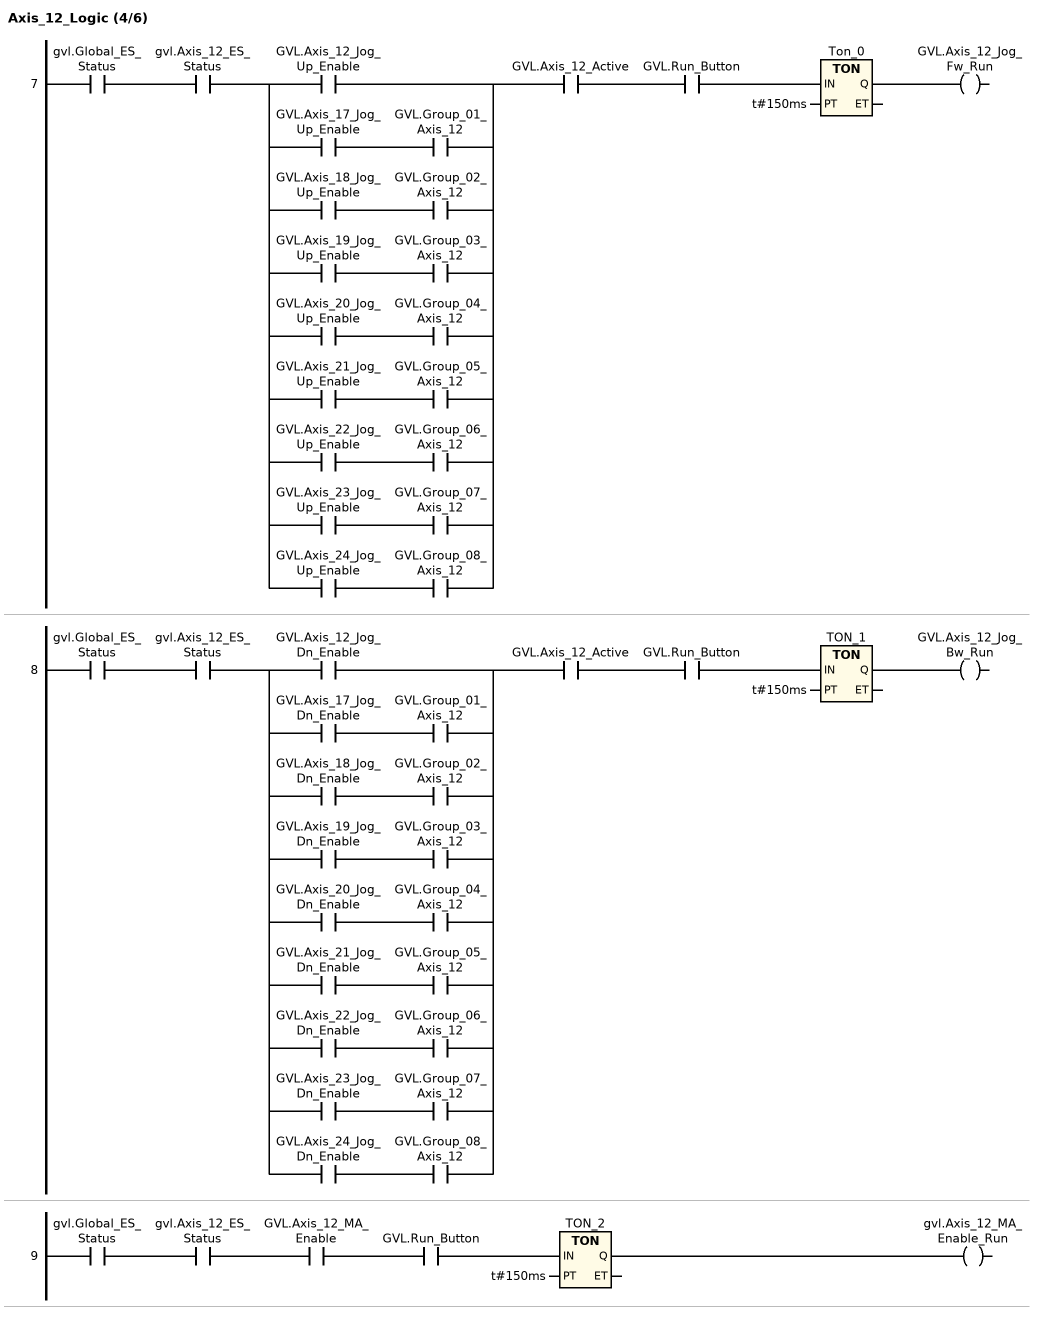
// NETWORK 7
Ton_0(IN := gvl.Global_ES_Status AND gvl.Axis_12_ES_Status AND (GVL.Axis_12_Jog_Up_Enable OR GVL.Axis_17_Jog_Up_Enable AND GVL.Group_01_Axis_12 OR GVL.Axis_18_Jog_Up_Enable AND GVL.Group_02_Axis_12 OR GVL.Axis_19_Jog_Up_Enable AND GVL.Group_03_Axis_12 OR GVL.Axis_20_Jog_Up_Enable AND GVL.Group_04_Axis_12 OR GVL.Axis_21_Jog_Up_Enable AND GVL.Group_05_Axis_12 OR GVL.Axis_22_Jog_Up_Enable AND GVL.Group_06_Axis_12 OR GVL.Axis_23_Jog_Up_Enable AND GVL.Group_07_Axis_12 OR GVL.Axis_24_Jog_Up_Enable AND GVL.Group_08_Axis_12) AND GVL.Axis_12_Active AND GVL.Run_Button, PT := t#150ms); // TON
GVL.Axis_12_Jog_Fw_Run := Ton_0.Q;

// NETWORK 8
TON_1(IN := gvl.Global_ES_Status AND gvl.Axis_12_ES_Status AND (GVL.Axis_12_Jog_Dn_Enable OR GVL.Axis_17_Jog_Dn_Enable AND GVL.Group_01_Axis_12 OR GVL.Axis_18_Jog_Dn_Enable AND GVL.Group_02_Axis_12 OR GVL.Axis_19_Jog_Dn_Enable AND GVL.Group_03_Axis_12 OR GVL.Axis_20_Jog_Dn_Enable AND GVL.Group_04_Axis_12 OR GVL.Axis_21_Jog_Dn_Enable AND GVL.Group_05_Axis_12 OR GVL.Axis_22_Jog_Dn_Enable AND GVL.Group_06_Axis_12 OR GVL.Axis_23_Jog_Dn_Enable AND GVL.Group_07_Axis_12 OR GVL.Axis_24_Jog_Dn_Enable AND GVL.Group_08_Axis_12) AND GVL.Axis_12_Active AND GVL.Run_Button, PT := t#150ms); // TON
GVL.Axis_12_Jog_Bw_Run := TON_1.Q;

// NETWORK 9
TON_2(IN := gvl.Global_ES_Status AND gvl.Axis_12_ES_Status AND GVL.Axis_12_MA_Enable AND GVL.Run_Button, PT := t#150ms); // TON
gvl.Axis_12_MA_Enable_Run := TON_2.Q;

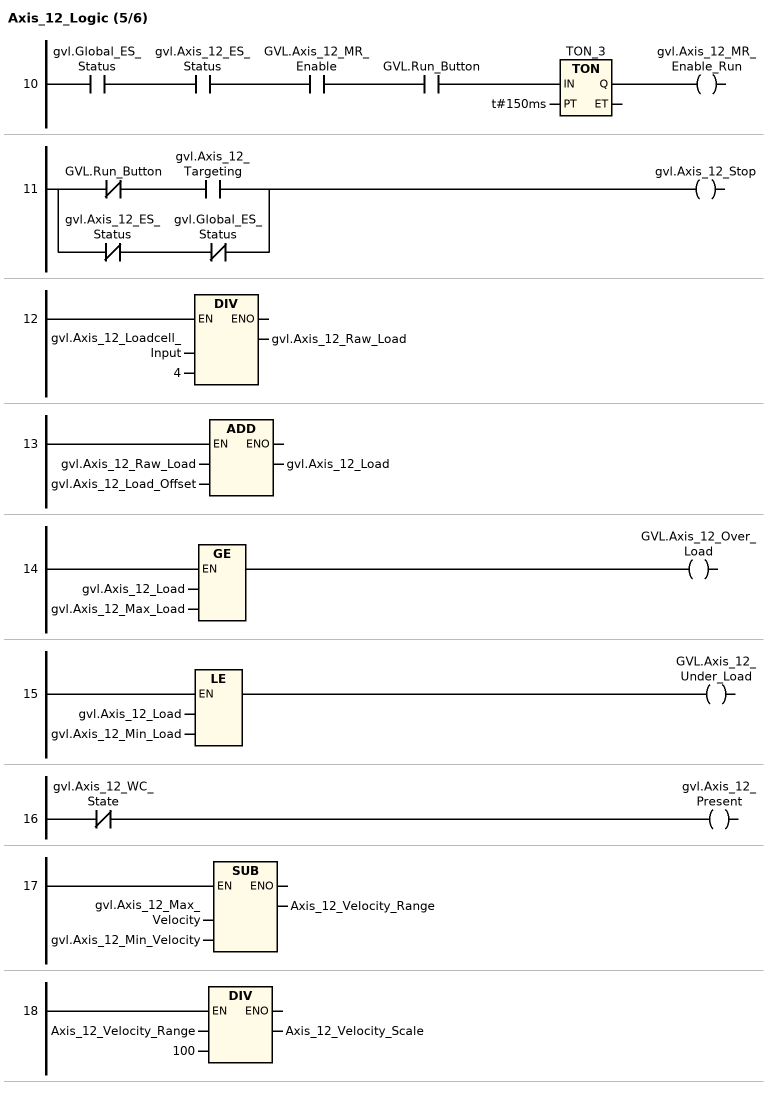
// NETWORK 10
TON_3(IN := gvl.Global_ES_Status AND gvl.Axis_12_ES_Status AND GVL.Axis_12_MR_Enable AND GVL.Run_Button, PT := t#150ms); // TON
gvl.Axis_12_MR_Enable_Run := TON_3.Q;

// NETWORK 11
gvl.Axis_12_Stop := NOT GVL.Run_Button AND gvl.Axis_12_Targeting OR NOT gvl.Axis_12_ES_Status AND NOT gvl.Global_ES_Status;

// NETWORK 12
gvl.Axis_12_Raw_Load := gvl.Axis_12_Loadcell_Input / 4;

// NETWORK 13
gvl.Axis_12_Load := gvl.Axis_12_Raw_Load + gvl.Axis_12_Load_Offset;

// NETWORK 14
GVL.Axis_12_Over_Load := gvl.Axis_12_Load >= gvl.Axis_12_Max_Load;

// NETWORK 15
GVL.Axis_12_Under_Load := gvl.Axis_12_Load <= gvl.Axis_12_Min_Load;

// NETWORK 16
gvl.Axis_12_Present := NOT gvl.Axis_12_WC_State;

// NETWORK 17
Axis_12_Velocity_Range := gvl.Axis_12_Max_Velocity - gvl.Axis_12_Min_Velocity;

// NETWORK 18
Axis_12_Velocity_Scale := Axis_12_Velocity_Range / 100;

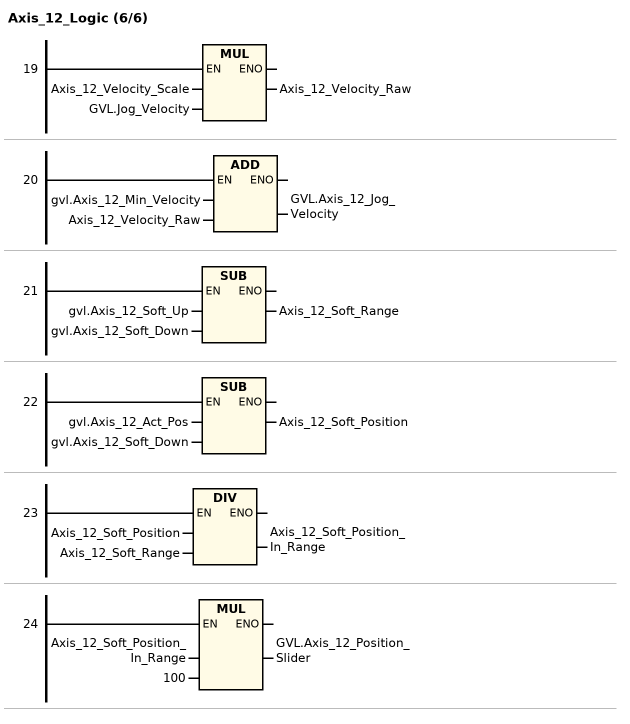
// NETWORK 19
Axis_12_Velocity_Raw := Axis_12_Velocity_Scale * GVL.Jog_Velocity;

// NETWORK 20
GVL.Axis_12_Jog_Velocity := gvl.Axis_12_Min_Velocity + Axis_12_Velocity_Raw;

// NETWORK 21
Axis_12_Soft_Range := gvl.Axis_12_Soft_Up - gvl.Axis_12_Soft_Down;

// NETWORK 22
Axis_12_Soft_Position := gvl.Axis_12_Act_Pos - gvl.Axis_12_Soft_Down;

// NETWORK 23
Axis_12_Soft_Position_In_Range := Axis_12_Soft_Position / Axis_12_Soft_Range;

// NETWORK 24
GVL.Axis_12_Position_Slider := Axis_12_Soft_Position_In_Range * 100;

END_PROGRAM

// ---- POUs/Axis_13_Function_Blocks.TcPOU
PROGRAM Axis_13_Function_Blocks
VAR
END_VAR

